% RSLogix 500 project LAB 3 SCAD BWFG_BAK102.RSS, saved by version 8.40.00.08 %
PROJECT "LAB2_BGJ"    % processor: SLC 500, 1747-L541 %

PROGRAM FILES
  LAD 2   2 rungs

DATA FILES
  O0 OUTPUT  68 elements
  I1 INPUT  68 elements
  S2 STATUS  164 elements
  B3 BINARY  10 elements
  T4 TIMER  51 elements
  C5 COUNTER  102 elements
  R6 CONTROL  1 elements
  N7 INTEGER  1 elements
  F8 FLOAT  1 elements

LADDER 2
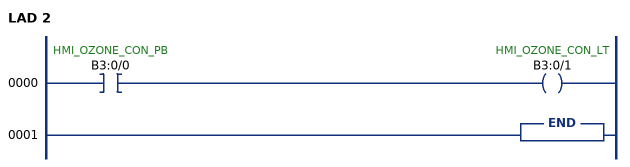
% Rung: 0 %
SOR XIC B3:0/0 OTE B3:0/1 EOR
%   B3:0/0  "HMI_OZONE_CON_PB" %
%   B3:0/1  "HMI_OZONE_CON_LT" %
% Rung: 1 %
SOR END EOR

OTHER DOCUMENTED ADDRESSES
  B3:0/2  "PART 2 START/STOP MEMORY CASCADED TIMERS"
  B3:0/3  "PART 3 START/STOP MEMORY"
  B3:0/10  "PART 1 START/STOP MEMORY"
  B3:1/4  "PART 2 START/STOP MEMORY CASCADED TIMERS"
  B3:1/14  "PART 3 START/STOP MEMORY"
  C5:1  "PART 3 UP/DOWN COUNTER"
  C5:1/CU  "COUNT UP ENABLED CTU IS ENERGIZED"
  C5:1/DN  "ACC IS GREATER THAN OR EQUAL TO PRE VALUE (25 IN THIS EXAMPLE)"
  C5:5  "PART 3 UP/DOWN COUNTER"
  C5:5.ACC  "SEND COUNTER ACCUMULATOR TO LED DISPLAY"
  C5:5.PRE  "LOAD COUNT PRESET FROM THUMBWHEEL"
  C5:10  "PART 3 UP/DOWN COUNTER"
  C5:10.ACC  "COUNTER ACC TO LED DISPLAY"
  C5:10.PRE  "LOAD COUNT PRESET FROM THUMBWHEEL"
  C5:10/CD  "CTD INSTRUCTION ENABLED"
  C5:10/CU  "CTU INSTRUCTION ENABLED"
  C5:10/DN  "COUNT ACC>=PRE (DONE)"
  C5:10/OV  "COUNTER ACC >32767 (OVERFLOW) ACC WRAPS TO ZERO"
  C5:10/UN  "COUNTER ACC LESS THAN -32768 ACC WRAPS TO ZERO"
  C5:31  "1ST COUNTER HORN ON TIME COUNTS 0.3 SEC (6 X 0.05 SEC)"
  C5:31/DN  "1ST COUNTER DONE ENGAGE 2ND COUNTER"
  C5:32  "2ND COUNTER HORN OFF TIME COUNTS 0.6 SEC (12 X 0.05 SEC)"
  C5:32/DN  "2ND COUNTER DONE RESET COUNTERS"
  C5:33  "PART 3 UP/DOWN COUNTER"
  C5:33.ACC  "DISPLAY UP/DOWN COUNTER ACC ON LED DISPLAY"
  C5:33.PRE  "LOAD UP/DOWN COUNTER PRESET FROM THUMBWHEEL"
  C5:33/DN  "UP/DOWN COUNTER DONE ENGAGE HORN"
  C5:34  "HORN CYCLE COUNTER STOP HORN AFTER 5 CYCLES"
  C5:100  "MINUTES FOR 24 HR CLOCK"
  C5:100.ACC  "DISPLAY MINUTES ON LED DISPLAY"
  C5:100/DN  "INDEX HOUR COUNTER EVERY 60 MINUTES"
  C5:101  "HOURS FOR 24 HR CLOCK"
  C5:101/DN  "RESET HOUR COUNT AT BEGINNING OF A NEW DAY"
  I:1.0/0  "1PBLT-BUTTON RESET COUNTER"
  I:1.0/1  "2PBLT BUTTON PART1: LOAD TIMER PART2: LOAD RED TIME PART3: LOAD HORN ON TIME"
  I:1.0/2  "3PBLT BUTTON PART 2: LOAD GREEN TIME PART 3: LOAD HORN OFF TIME"
  I:1.0/3  "4PBLT BUTTON PART 2: LOAD AMBER TIME PART3: LOAD COUNTER PRESET"
  I:1.0/4  "5PB START BUTTON"
  I:1.0/5  "6PB COUNT UP"
  I:1.0/6  "7PB STOP BUTTON"
  I:1.0/7  "8PB STOP BUTTON"
  I:1.0/8  "COUNT UP PB"
  I:1.0/9  "COUNT DOWN PB"
  I:1.0/10  "3SS POS 1 POSITION"
  I:1.0/11  "3SS POS 3 POSITION"
  I:1.0/12  "SET MINUTES FROM THUMBWHELL WHEN PRESSED"
  I:1.0/13  "SET HOURS FROM THUMBWHEEL WHEN PRESSED"
  I:1.0/14  "SHOW SECONDS ON LED DISPLAY"
  I:1.0/15  "SHOW MINUTES ON LED DISPLAY"
  I:3.0  "LOAD ACCUMULATOR FROM THUMBWHEEL"
  I:5.0/0  "SHOW HOURS ON LED DISPLAY"
  O:2.0/0  "GREEN LIGHT"
  O:2.0/1  "AMBER LIGHT"
  O:2.0/2  "RED LIGHT"
  O:2.0/3  "FLASHING LIGHT"
  O:2.0/4  "1LT GREEN LIGHT"
  O:2.0/5  "2LT FLASHING LIGHT"
  O:2.0/6  "3LT RED LIGHT FLASH ON/OFF"
  O:2.0/7  "4LT GREEN STACK LIGHT"
  O:2.0/8  "5LT AMBER STACK LIGHT"
  O:2.0/9  "6LT RED STACK LIGHT"
  O:2.0/10  "1AH HORN"
  O:2.0/11  "COUNTER UNDERFLOW"
  O:4.0  "ACCUMULATOR TO LED DISPLAY"
  T4:1  "FREE RUNNING TIMER"
  T4:1.ACC  "DISPLAY TIMER ACC ON LED DISPLAY"
  T4:1.ACC/6  "0.64 SEC FLASHING BIT OF FREE RUN TIMER"
  T4:1.PRE  "LOAD FREE RUN TIMER FROM THUMBWHEEL"
  T4:1/DN  "TIMER DONE RESET FREE-RUN"
  T4:2  "STAGE 1 TIMER FOR CASCADED TIMING CIRCUIT"
  T4:2/DN  "STAGE 1 DONE ENABLE STAGE 2"
  T4:2/TT  "O.75 SEC FLASHER WHILE STAGE 1 IS TIMING"
  T4:3  "STAGE 2 TIMER FOR CASCADED TIMING CIRCUIT"
  T4:3/DN  "LAST TIMER DONE RESET CIRCUIT FOR NEXT CYCLE"
  T4:4  "GREEN LIGHT TIMER"
  T4:4/DN  "GREEN TIME DONE START AMBER TIME"
  T4:5  "AMBER LIGHT TIMER"
  T4:5/DN  "AMBER TIME DONE START RED"
  T4:6  "RED LIGHT TIMER"
  T4:6/DN  "RED TIME DONE RESET FOR NEXT CYCLE"
  T4:10  "PART 1 FREE RUN TIMER"
  T4:10.ACC  "PART 1 FREE RUN TIMER TO LED DISPLAY"
  T4:10.PRE  "LOAD FREE RUN TIMER FROM THUMBWHEEL"
  T4:10/DN  "FREE RUN TIMER DONE RESET FOR NEXT CYCLE"
  T4:11  "PART 1 FREE RUNNING TIMER"
  T4:11.ACC  "DISPLAY TIMER ACC ON LED DISPLAY"
  T4:11.ACC/5  "0.32 SEC FLASHER"
  T4:11.ACC/6  "0.32 SEC FLASHER"
  T4:11.PRE  "LOAD FREE RUN TIMER PREST FROM THUMBWHEEL"
  T4:11/DN  "TIMER DONE RESET"
  T4:12  "PART 2 GREEN LIGHT CASCADE TIMER 2"
  T4:12.PRE  "LOAD GREEN TIME PRESET FROM THUMBWHEEL"
  T4:12/DN  "GREEN LIGHT TIMER DONE"
  T4:12/TT  "GREEN LIGHT TIMER TIMING"
  T4:13  "PART 2 AMBER LIGHT CASCADE TIMER 3"
  T4:13.PRE  "LOAD AMBER TIME PRESET FROM THUMBWHEEL"
  T4:13/DN  "LAST CASCADE TIMER DONE RESET CYCLE"
  T4:13/TT  "AMBER LIGHT TIMER TIMING"
  T4:20  "PART 3 HORN TIMER 2.25 SEC"
  T4:20/DN  "HORN TIME DONE"
  T4:21  "PART 2 RED LIGHT TIME CASCADED TIMER 1"
  T4:21.PRE  "LOAD RED TIME PRESET FROM THUMBWHEEL"
  T4:21/DN  "RED TIME DONE START GREEN TIMER"
  T4:21/TT  "ENERGIZE RED LIGHT"
  T4:22  "PART 2 GREEN LIGHT CASCADE TIMER 2"
  T4:22.PRE  "LOAD GREEN TIME PRESET FROM THUMBWHEEL"
  T4:22/DN  "GREEN TIME DONE START AMBER TIMER"
  T4:22/TT  "ENERGIZE GREEN LIGHT"
  T4:23  "PART 2 AMBER LIGHT CASCADE TIMER 3"
  T4:23.PRE  "LOAD AMBER TIME PRESET FROM THUMBWHEEL"
  T4:23/DN  "LAST CASCADE TIMER DONE RESET CYCLE"
  T4:23/TT  "ENERGIZE AMBER LIGHT"
  T4:24  "LIGHT ON TIME"
  T4:24/DN  "1ST CASCADE TIME DONE START 2ND TIMER"
  T4:24/TT  "LIGHT ON TIME"
  T4:25  "LIGHT OFF TIME"
  T4:25/DN  "2ND CASCADE TIMER DONE RESET CIRCUIT"
  T4:30  "PART 3 HORN TIMER 2.75 SEC"
  T4:30/DN  "HORN TIME DONE SHUT OFF HORN"
  T4:31  "0.05 SEC FREE RUN TIMER"
  T4:31/DN  "TIME DONE RESET FREE RUN TIMER AND INDEX COUNTER"
  T4:32  "HORN ON TIME"
  T4:32.PRE  "LOAD HORN ON TIME FROM THUMBWHEEL"
  T4:32/DN  "HORN ON TIME DONE"
  T4:33  "HORN OFF TIME"
  T4:33.PRE  "LOAD HORN OFF TIME FROM THUBWHEEL"
  T4:33/DN  "HORN OFF TIME DONE RESET TIMERS"
  T4:50  "SECONDS FOR 24 HR CLOCK"
  T4:50/DN  "RESET FREE RUN TIMER"

OTHER INSTRUCTION COMMENTS
  C5:100.ACC FRD  "MINUTES FOR 24 HR CLOCK"
  C5:101 RES  "RESET HOUR COUNT START OF NEW DAY"
  C5:100 RES  "RESET MINUTE COUNT EVERY HOUR"
  T4:50/DN XIC  "INDEX MINUTE COUNTER EVERY 60 SECONDS"
  C5:10 RES  "PART 3 RESET COUNTER TO ZERO"
  C5:1 RES  "PART 3 RESET COUNTER TO ZERO"

COMMENTS NOT ATTACHED TO A CURRENT RUNG
  T4:2: CASCADED TIMER CIRCUIT CONSISTING OF TWO TIMING STAGES WITH T4:2 AND T4:3
  O:2.0/3: FLASHING LIGHT FROM ACC BIT OF FREE RUNNING TIMER
  T4:1: FREE RUNNING TIMER CIRCUIT
  B3:0/0: PAGE TITLE TO START INTERNAL MEMORY BIT ON A NEW PAGE WHEN PRINTING / INTERNAL MEMORY BIT B3/0 FROM FILE B3 - RUNG COMMENT
  B3:0/10: PART 1 - FREE RUN TIMER PLUS THUMBWHEEL AND LED DISPLAY / Lab Solution - Brent Brooks - Winter 2008
  B3:1/4: PART 2 - CASCADED TIMERS AND SIMPLE TRAFFIC LIGHT
  B3:1/14: PART 3 - HORN TIMER AND UP/DOWN COUNTER, THUMBWHEEL AND LED DISPLAY
  B3:0/3: PART 3 - HORN TIMER AND UP/DOWN COUNTER AND THUMBWHEEL AND LED DISPLAY
  B3:0/2: PART 2 - CASCADED TIMERS AND TRAFFIC LIGHT

DATA TABLE (non-zero values as saved)
DATA B3
% B3:0 % 0X0000 0X4000 0X0000 0X0000 0X0000 0X0000 0X0000 0X0000 0X0000 0X0000
DATA T4
% .PRE .ACC %
% T4:1 % 1500 0
% T4:2 % 75 0
% T4:3 % 150 0
% T4:4 % 15 0
% T4:5 % 5 0
% T4:6 % 20 0
% T4:10 % 1500 0
% T4:11 % 128 0
% T4:12 % 500 0
% T4:13 % 200 0
% T4:20 % 225 0
% T4:21 % 525 0
% T4:22 % 245 0
% T4:23 % 175 0
% T4:24 % 75 0
% T4:25 % 50 0
% T4:30 % 275 0
% T4:31 % 5 0
% T4:32 % 25 25
% T4:33 % 150 30
% T4:50 % 60 0
DATA C5
% .PRE .ACC %
% C5:1 % 25 0
% C5:5 % 25 0
% C5:10 % 25 0
% C5:31 % 6 1
% C5:32 % 12 0
% C5:33 % 10 10
% C5:34 % 6 6
% C5:100 % 60 35
% C5:101 % 24 10
